(* Logix 5000 project; controller boca_de_pescado Emulate 5570 rev 32.11; software revision 32.00 *)

TASK MainTask (continuous, watchdog 500 ms) : MainProgram

MODULES
   Local : Emulate 5570 (ICP 2, rev 32.11)
      I_O : vendor 1 type 0 code 15 (ICP 3, rev 1.1, Output RPI 50 ms)   // Señales de entrada y salida
END_MODULES

VAR_GLOBAL   (* controller tags *)
   S1 : ALIAS FOR Local:3:I.Data[1].0;
   S2 : ALIAS FOR Local:3:I.Data[1].1;
   S3 : ALIAS FOR Local:3:I.Data[1].2;
   S4 : ALIAS FOR Local:3:I.Data[1].3;
   S5 : ALIAS FOR Local:3:I.Data[1].4;
   S6 : ALIAS FOR Local:3:I.Data[1].5;
   Start : ALIAS FOR Local:3:I.Data[1].6;
   Stop : ALIAS FOR Local:3:I.Data[1].7;
   Y1 : ALIAS FOR Local:3:O.Data[0].0;
   Y2 : ALIAS FOR Local:3:O.Data[0].1;
   Y3 : ALIAS FOR Local:3:O.Data[0].2;
   Y4 : ALIAS FOR Local:3:O.Data[0].3;
   Y5 : ALIAS FOR Local:3:O.Data[0].4;
   Y6 : ALIAS FOR Local:3:O.Data[0].5;
END_VAR

PROGRAM MainProgram   (* main routine MainRoutine *)
VAR
   Action_000 : SFC_ACTION := (Status := 16#0020_0000, PauseTimer := 1);
   Action_001 : SFC_ACTION := (Status := 16#0020_0000, PauseTimer := 1);
   Action_002 : SFC_ACTION := (Status := 16#0020_0000, PauseTimer := 1);
   Action_003 : SFC_ACTION := (Status := 16#0020_0000, PauseTimer := 1);
   Action_004 : SFC_ACTION := (Status := 16#0020_0000, PauseTimer := 1);
   Action_005 : SFC_ACTION := (Status := 16#0020_0000, PauseTimer := 1);
   Action_006 : SFC_ACTION := (Status := 16#0020_0000, PauseTimer := 1);
   Action_007 : SFC_ACTION := (Status := 16#0020_0000, PauseTimer := 1);
   Action_008 : SFC_ACTION := (Status := 16#0020_0000, PauseTimer := 1);
   Action_009 : SFC_ACTION := (Status := 16#0020_0000, PauseTimer := 1);
   Step_000 : SFC_STEP := (Status := 16#0020_0000, PauseTimer := 1);
   Step_001 : SFC_STEP := (Status := 16#0020_0000, PauseTimer := 1, PRE := 2000);
   Step_002 : SFC_STEP := (Status := 16#0020_0000, PauseTimer := 1, PRE := 2000);
   Step_003 : SFC_STEP := (Status := 16#0020_0000, PauseTimer := 1, PRE := 50);
   Step_004 : SFC_STEP := (Status := 16#0020_0000, PauseTimer := 1);
   Step_005 : SFC_STEP := (Status := 16#0020_0000, PauseTimer := 1);
   Step_006 : SFC_STEP := (Status := 16#0020_0000, PauseTimer := 1);
   Step_007 : SFC_STEP := (Status := 16#0020_0000, PauseTimer := 1);
   Step_008 : SFC_STEP := (Status := 16#0020_0000, PauseTimer := 1);
   Step_009 : SFC_STEP := (Status := 16#0020_0000, PauseTimer := 1, PRE := 5000);
   Step_010 : SFC_STEP := (Status := 16#0020_0000, PauseTimer := 1);
   Tran_000 : BOOL;
   Tran_001 : BOOL;
   Tran_002 : BOOL;
   Tran_003 : BOOL;
   Tran_004 : BOOL;
   Tran_005 : BOOL;
   Tran_006 : BOOL;
   Tran_007 : BOOL;
   Tran_008 : BOOL;
   Tran_009 : BOOL;
   Tran_010 : BOOL;
   Tran_011 : BOOL;
   Tran_012 : BOOL;
END_VAR

ROUTINE graphcet   (* sequential function chart *)
// descripción en graphcet de la rutina
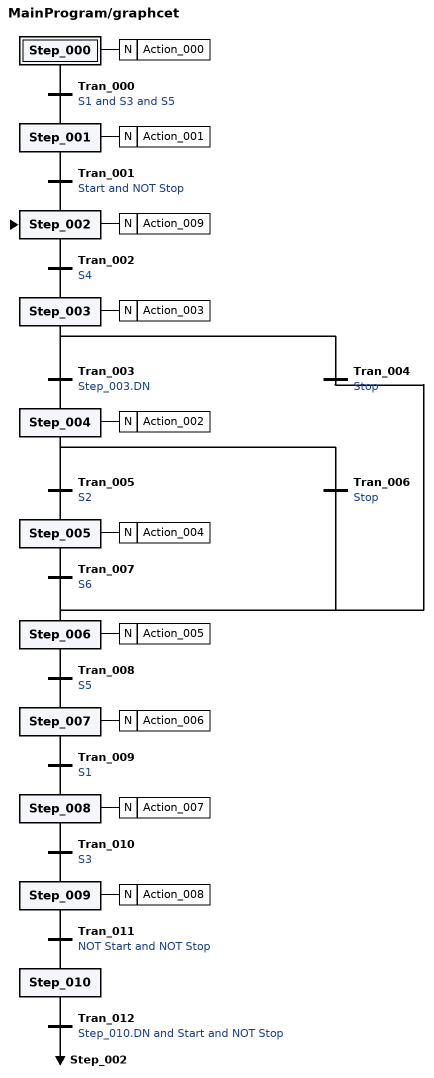
   INITIAL_STEP Step_000:
      ACTION Action_000 (N):
         Y1:=1;
         Y2:=0;
         Y3:=1;
         Y4:=0;
         Y5:=1;
         Y6:=0;
      END_ACTION
   END_STEP
   TRANSITION Tran_000 FROM Step_000 TO Step_001
      := S1 and S3 and S5
   END_TRANSITION
   STEP Step_001:
      ACTION Action_001 (N):
         Y1:=0;
         Y3:=0;
         Y5:=0;
      END_ACTION
   END_STEP
   TRANSITION Tran_001 FROM Step_001 TO Step_002
      := Start and NOT Stop
   END_TRANSITION
   STEP Step_002:
      ACTION Action_009 (N):
         Y4:=1;
      END_ACTION
   END_STEP
   TRANSITION Tran_002 FROM Step_002 TO Step_003
      := S4
   END_TRANSITION
   STEP Step_003:
      ACTION Action_003 (N):
         Y4:=0;
      END_ACTION
   END_STEP
   TRANSITION Tran_003 FROM Step_003 TO Step_004
      := Step_003.DN
   END_TRANSITION
   STEP Step_004:
      ACTION Action_002 (N):
         Y2:=1;
      END_ACTION
   END_STEP
   TRANSITION Tran_005 FROM Step_004 TO Step_005
      := S2
   END_TRANSITION
   STEP Step_005:
      ACTION Action_004 (N):
         Y2:=0;
         Y6:=1;
      END_ACTION
   END_STEP
   TRANSITION Tran_007 FROM Step_005 TO Step_006
      := S6
   END_TRANSITION
   TRANSITION Tran_006 FROM Step_004 TO Step_006
      := Stop
   END_TRANSITION
   TRANSITION Tran_004 FROM Step_003 TO Step_006
      := Stop
   END_TRANSITION
   STEP Step_006:
      ACTION Action_005 (N):
         Y6:=0;
         Y5:=1;
      END_ACTION
   END_STEP
   TRANSITION Tran_008 FROM Step_006 TO Step_007
      := S5
   END_TRANSITION
   STEP Step_007:
      ACTION Action_006 (N):
         Y5:=0;
         Y1:=1;
      END_ACTION
   END_STEP
   TRANSITION Tran_009 FROM Step_007 TO Step_008
      := S1
   END_TRANSITION
   STEP Step_008:
      ACTION Action_007 (N):
         Y1:=0;
         Y3:=1;
      END_ACTION
   END_STEP
   TRANSITION Tran_010 FROM Step_008 TO Step_009
      := S3
   END_TRANSITION
   STEP Step_009:
      ACTION Action_008 (N):
         Y3:=0;
      END_ACTION
   END_STEP
   TRANSITION Tran_011 FROM Step_009 TO Step_010
      := NOT Start and NOT Stop
   END_TRANSITION
   STEP Step_010:
   END_STEP
   TRANSITION Tran_012 FROM Step_010 TO Step_002
      := Step_010.DN and Start and NOT Stop
   END_TRANSITION
END_ROUTINE

ROUTINE MainRoutine   (* ladder *)
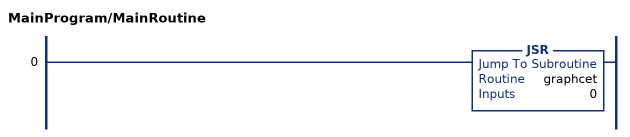
   0: JSR(graphcet,0);
END_ROUTINE
END_PROGRAM
